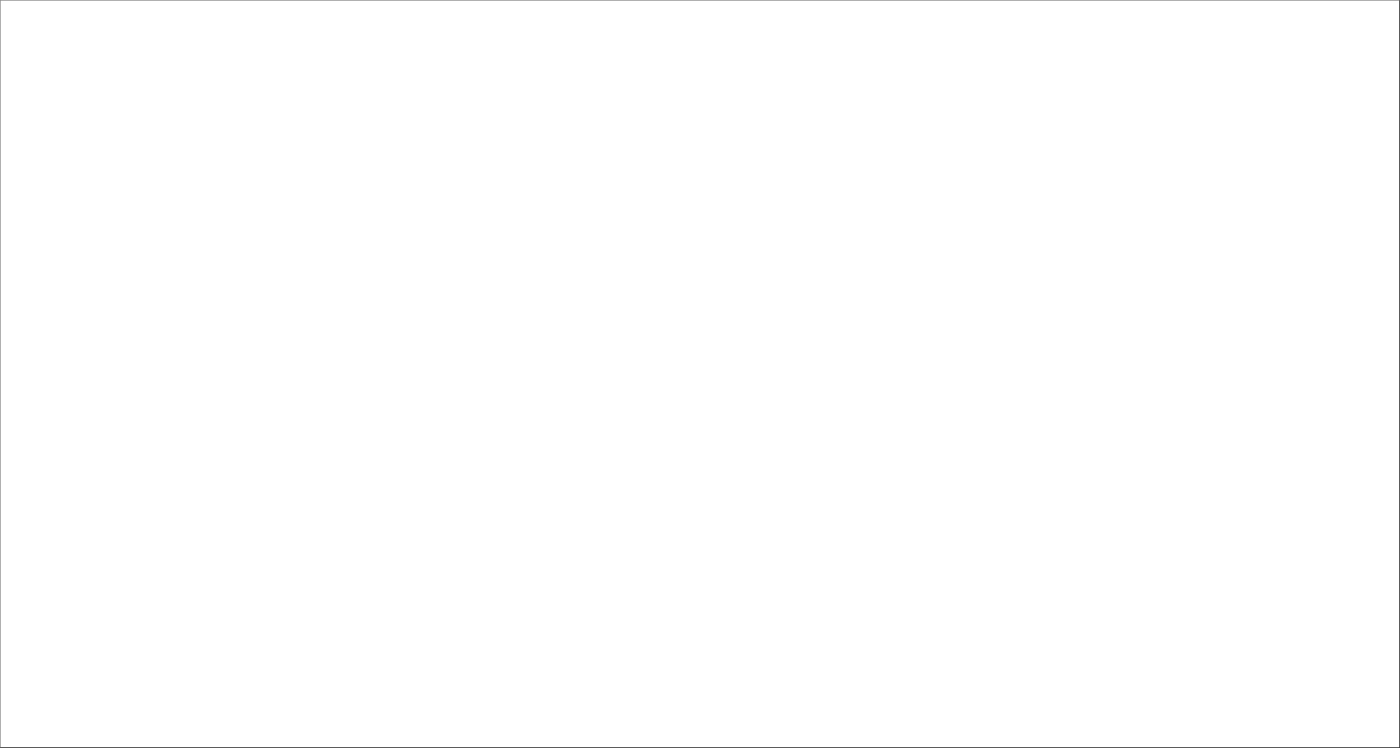
VISUALIZATION Farbverlauf  // 2438x1304
    Rectangle (0,0 2438x1304)
END_VISUALIZATION

(* stored: Version 1.1.0.1, ProductVersion 3.1.4024.3
   Visu Farbverlauf: Id {4c8763b5-16b3-41d2-a1bd-7ddb08afc057} *)
